PROGRAM MAIN
VAR
	nPmeter AT %I* : INT;
	nScaledMax AT %Q* : INT := 15;
	nValue AT %Q* : INT;
END_VAR

//Lees de potentiometer in en verschaal deze waarden naar een getal tussen 0 en de variable nScaledMax. Geef voorlopig de initial value van 10 mee.

nValue := REAL_TO_BYTE(nPmeter/32767.0 * nScaledMax);

END_PROGRAM

(* stored: Version 1.1.0.1, ProductVersion 3.1.4024.12
   POU MAIN: Id {b3a14c7f-10c1-45f8-9040-3332cea8f9f6}, SpecialFunc None *)
